// TwinCAT 3 PLC project VibrodriverPLC
// ProgramVersion: 3.1.4024.0
// libraries:
//   Tc2_MC2, * (Beckhoff Automation GmbH)
//   Tc2_NC, * (Beckhoff Automation GmbH)
//   Tc2_Standard, * (Beckhoff Automation GmbH)
//   Tc2_System, * (Beckhoff Automation GmbH)
//   Tc2_Utilities, * (Beckhoff Automation GmbH)
//   Tc3_Module, * (Beckhoff Automation GmbH)
//   VisuDialogs, * (System)
//   VisuSymbols,3.5.10.0,System
// project tree:
//   / GlobalTextList.TcGTLO, PlcTask.TcTTO, Visualization Manager.TcVMO (not stored)
//   POUs/ MAIN.TcPOU, FB_ReadGeophone.TcPOU, FB_ReadAccelerometer.TcPOU (not stored), P_ReadSensors.TcPOU (not stored)
//   VISUs/ hmi.TcVIS

CONFIGURATION VibrodriverPLC
    RESOURCE PLC ON TwinCAT3
        TASK PlcTask(INTERVAL := T#10ms, PRIORITY := 20);
        PROGRAM MAIN WITH PlcTask : MAIN;
        PROGRAM P_ReadSensors WITH PlcTask : P_ReadSensors;
    END_RESOURCE
END_CONFIGURATION

// ---- POUs/MAIN.TcPOU
PROGRAM MAIN
VAR

	bRun : BOOL := FALSE; // main control	

	axes : ARRAY[0..3] OF AXIS_REF; // [BL BR TL TR] (linked in MOTION)
	
	// motion control function blocks
	arrMCResets        		: ARRAY[0..3] OF MC_Reset;
	arrMCPowers				: ARRAY[0..3] OF MC_Power;
	arrMCSetPositions		: ARRAY[0..3] OF MC_SetPosition;
	arrMCMoveAbsolutes		: ARRAY[0..3] OF MC_MoveAbsolute;
	arrMCMoveRelatives		: ARRAY[0..3] OF MC_MoveRelative;
	arrMCMoveVelocitys 		: ARRAY[0..3] OF MC_MoveVelocity;
	arrMCHalts				: ARRAY[0..3] OF MC_Halt;
	arrMCGearIns			: ARRAY[1..3] OF MC_GearIn;
	arrMCGearOuts			: ARRAY[1..3] OF MC_GearOut;
	arrMCPhaseAbsolutes     : ARRAY[1..3] OF MC_PhasingAbsolute;
	
	arrRelsDone : ARRAY[0..3] OF BOOL; // keep track of if each motor is done its relative movement
	arrRelsDoneZero : ARRAY[0..3] OF BOOL; // keep track of if each motor is done its relative movement
	arrMCMoveRelativesZero	: ARRAY[0..3] OF MC_MoveRelative;
	arrZeroPoss : ARRAY[0..3] OF LREAL;
	
	arrHexErrors : ARRAY[0..3] OF T_MaxString; // store hex format of axes errors
	
	i: INT; // generic loop index 1
	j: INT; // generic loop index 2
	k: INT; // generic loop index 3
	
	bStarted : BOOL := FALSE; // if started is complete
	bCoupled : BOOL := FALSE;
	iMode : INT := 2; // 0 = move abs, 1 = move rel, 2 = move vel, 3 = zero nearest
	
	// button bools
	bStart  : BOOL := FALSE;
	bStop   : BOOL := TRUE;
	bCouple : BOOL := FALSE;
	bAbsPos : BOOL := FALSE;
	bRelPos	: BOOL := FALSE;
	bVel	: BOOL := TRUE;
	
	// taps
	bZeroNear : BOOL := FALSE;
	bResetFaults :BOOL := FALSE;
	
	// values in HMI
	iPos : INT := 0;
	iVel : INT := 1440;
	iAcc : INT := 720;
	iPhs : INT := 0;
	
	// track previous values for updating function blocks
	iPrevPos : INT := iPos;
	iPrevVel : INT := iVel;
	iPrevAcc : INT := iAcc;
	iPrevPhs : INT := iPhs;
	
	iMaxVel : INT := 3600; // max 10 hz
	eDirec : MC_Direction := MC_Direction.MC_Negative_Direction;
	iDirMult : INT := -1; // multiplier: actVel = setVel * mult (used to reverse default)
	
	// outside first and last are ignored
	iFirstIdx : INT := 2; // first motor index to control
	iLastIdx : INT := 3; // last motor index to control
	
	iEndIdx : INT := 3; // used to ignore other indices when the motors are coupled, set such that only the iFirstIdx index motor is controlled 
END_VAR

// test
FOR i := iFirstIdx TO iLastIdx DO
	// UPDATE AXES STATUS
	axes[i].ReadStatus();
	// UPDATE HEX ERRORS
	arrHexErrors[i] := WORD_TO_HEXSTR(in:=UDINT_TO_WORD(MAIN.axes[i].Status.ErrorID), iPrecision:=4, bLoCase:=FALSE);
	// RESTRICT VELOCITY
	IF ABS(axes[i].NcToPlc.ActVelo) > iMaxVel THEN
		M_SetState(0);
	END_IF
END_FOR


// STARTUP
// <<<<<<<<<<<<<<<<<<<<<<<<<<<<<<<<<<<<<<<<<<<<<<<<<<<<<<<
IF NOT bStarted THEN
	// start each motor
	FOR i := iFirstIdx TO iLastIdx DO
		// default to OFF despite variable values
		M_SetState(0);
		arrMCResets[i](Axis:=axes[i]);
		arrMCPowers[i](Axis:=axes[i], Enable:= TRUE, Enable_Positive:=TRUE, Enable_Negative:=TRUE);
	END_FOR
	
	// if all motors powered, set to started
	FOR i:=iFirstIdx TO iLastIdx DO
		IF NOT arrMCPowers[i].Status THEN
			EXIT;
		ELSIF i=iLastIdx THEN
			bStarted := TRUE;
			M_SetMode(2);
		END_IF
	END_FOR
END_IF
// >>>>>>>>>>>>>>>>>>>>>>>>>>>>>>>>>>>>>>>>>>>>>>>>>>>>>>>


// MODE SELECTION
// <<<<<<<<<<<<<<<<<<<<<<<<<<<<<<<<<<<<<<<<<<<<<<<<<<<<<<<
// prevent no mode selection
IF NOT bAbsPos AND iMode = 0 THEN
	bAbsPos := TRUE;
ELSIF NOT bRelPos AND iMode = 1 THEN
	bRelPos := TRUE;
ELSIF NOT bVel AND iMode = 2 THEN
	bVel := TRUE;
END_IF

// switch modes
IF iMode = 3 THEN
	M_SetMode(3);
ELSIF iMode = 4 THEN
	M_SetMode(4);
ELSIF bAbsPos AND iMode <> 0 THEN
	M_SetMode(0);
ELSIF bRelPos AND iMode <> 1 THEN
	M_SetMode(1);
ELSIF bVel AND iMode <> 2 THEN
	M_SetMode(2);
END_IF
// >>>>>>>>>>>>>>>>>>>>>>>>>>>>>>>>>>>>>>>>>>>>>>>>>>>>>>>


// RUN STATE SELECTION
// <<<<<<<<<<<<<<<<<<<<<<<<<<<<<<<<<<<<<<<<<<<<<<<<<<<<<<<
// prevent turning off a button, only swapping allowed
IF bRun AND NOT bStop THEN
	bStart := TRUE;
ELSIF NOT bRun AND NOT bStart THEN
	bStop := TRUE;
ELSE // invalid state
	bStop := TRUE;
END_IF

// on off logic
IF NOT bRun AND bStart THEN
	M_SetState(1);
END_IF
IF bStop THEN
	M_SetState(0);
END_IF

// handle zeroing button
IF bZeroNear AND NOT bRun THEN
	M_SetState(1);
	M_SetMode(3);
ELSIF bResetFaults AND NOT bRun THEN
	M_SetState(0);
	M_SetMode(4);
END_IF
// >>>>>>>>>>>>>>>>>>>>>>>>>>>>>>>>>>>>>>>>>>>>>>>>>>>>>>>


// COUPLING
// <<<<<<<<<<<<<<<<<<<<<<<<<<<<<<<<<<<<<<<<<<<<<<<<<<<<<<<
// disallow coupling while in motion
IF bCouple AND NOT bCoupled THEN
	FOR i:=iFirstIdx TO iLastIdx DO
		IF axes[i].Status.Moving THEN
			bCouple := FALSE;
			EXIT;
		END_IF
	END_FOR
END_IF

// COUPLE/UNCOUPLE GEARS
//arrMCGearOuts[1](Slave:=axes[1], Execute:=NOT bCouple AND bCoupled);
//arrMCGearOuts[2](Slave:=axes[2], Execute:=NOT bCouple AND bCoupled);
arrMCGearOuts[3](Slave:=axes[3], Execute:=NOT bCouple AND bCoupled);
//arrMCGearIns[1](Master:=axes[0], Slave:=axes[1], Execute:=bCouple AND NOT bCoupled, RatioNumerator:=-1);
//arrMCGearIns[2](Master:=axes[0], Slave:=axes[2], Execute:=bCouple AND NOT bCoupled, RatioNumerator:=-1);
arrMCGearIns[3](Master:=axes[2], Slave:=axes[3], Execute:=bCouple AND NOT bCoupled, RatioNumerator:=-1);

// check if uncoupling done
IF (NOT bCouple AND bCoupled)THEN
	FOR i:=iFirstIdx+1 TO iLastIdx DO
		IF NOT arrMCGearOuts[i].Done THEN
			EXIT;
		ELSIF i=iLastIdx THEN
			// if all out of gear, set the end index to the last index so that all the motors are controlled seperately again
			iEndIdx := iLastIdx;
			bCoupled := TRUE;
		END_IF;
	END_FOR
END_IF
// check if coupling done
IF (bCouple AND NOT bCoupled) THEN
	FOR i:=iFirstIdx+1 TO iLastIdx DO
		IF NOT arrMCGearIns[i].InGear THEN
			EXIT;
		ELSIF i=iLastIdx THEN
			// if all in gear, set the end index to the first index so that only the master is controlled
			iEndIdx := iFirstIdx;
			bCoupled := TRUE;
		END_IF;
	END_FOR
END_IF
// >>>>>>>>>>>>>>>>>>>>>>>>>>>>>>>>>>>>>>>>>>>>>>>>>>>>>>>





// operations to do only after startup
IF bStarted THEN
	

	// PHASING
	// set phase, master = BL, slave = TL
	// <<<<<<<<<<<<<<<<<<<<<<<<<<<<<<<<<<<<<<<<<<<<<<<<<<<<<<<
	
	IF iPrevPhs <> iPhs THEN
		//arrMCPhaseAbsolutes[1](Master:=axes[0], Slave:=axes[1], Execute:=FALSE); // set phase of BR w BL
		//arrMCPhaseAbsolutes[2](Master:=axes[0], Slave:=axes[2], Execute:=FALSE); // set phase of top w bottom
		arrMCPhaseAbsolutes[3](Master:=axes[2], Slave:=axes[3], Execute:=FALSE); // set phase of TR w TL
		iPrevPhs := iPhs;
	END_IF
	
	IF bRun AND bCoupled THEN
		// set phase of BR w BL
		//arrMCPhaseAbsolutes[1](Master:=axes[0], Slave:=axes[1], Execute:=TRUE, PhaseShift:=0, Velocity:=iVel+180);
		// set phase of top w bottom
		//arrMCPhaseAbsolutes[2](Master:=axes[0], Slave:=axes[2], Execute:=TRUE, PhaseShift:=iPhs, Velocity:=iVel+180);
		// set phase of TR w TL
		arrMCPhaseAbsolutes[3](Master:=axes[2], Slave:=axes[3], Execute:=TRUE, PhaseShift:=0, Velocity:=iVel+180);
	END_IF
	// >>>>>>>>>>>>>>>>>>>>>>>>>>>>>>>>>>>>>>>>>>>>>>>>>>>>>>>
	
	
	
	
	// MAIN COMMAND LOOP
	FOR i := iFirstIdx TO iEndIdx DO
		
	
		// CHANGE RESETING
		// <<<<<<<<<<<<<<<<<<<<<<<<<<<<<<<<<<<<<<<<<<<<<<<<<<<<<<<
		
		// if values have been updated, unexecute relevant functions so that they can restart with correct values
		IF (iPrevVel <> iVel) OR (iPrevAcc <> iAcc) THEN
			arrMCMoveAbsolutes[i](Axis:=axes[i], Execute:=FALSE);
			arrMCMoveRelatives[i](Axis:=axes[i], Execute:=FALSE);
			arrMCMoveVelocitys[i](Axis:=axes[i], Execute:=FALSE);
		ELSIF iPrevPos <> iPos THEN
			arrMCMoveAbsolutes[i](Axis:=axes[i], Execute:=FALSE);
			arrMCMoveRelatives[i](Axis:=axes[i], Execute:=FALSE);
		END_IF
		
		// if end index then set the previous values for change checks above ^
		IF i = iEndIdx THEN
			iPrevPos := iPos;
			iPrevVel := iVel;
			iPrevAcc := iAcc;
		END_IF
		// >>>>>>>>>>>>>>>>>>>>>>>>>>>>>>>>>>>>>>>>>>>>>>>>>>>>>>>
		
		
		// RELATIVE MOVEMENT OPERATION
		// <<<<<<<<<<<<<<<<<<<<<<<<<<<<<<<<<<<<<<<<<<<<<<<<<<<<<<<
		
		// check if relative movement is done, set to stop
		IF arrMCMoveRelatives[i].Done  THEN
			arrRelsDone[i] := TRUE;
			FOR j := iFirstIdx TO iEndIdx DO
				IF arrRelsDone[j] = FALSE THEN EXIT; END_IF
				IF j = iEndIdx THEN
					M_SetState(0);
					FOR k := iFirstIdx TO iLastIdx DO
						arrRelsDone[k] := FALSE;
					END_FOR
				END_IF
			END_FOR
		END_IF
		// check if relative movement is done, set to stop (SPECIFIC FOR ZEROING)
		IF arrMCMoveRelativesZero[i].Done  THEN
			arrRelsDoneZero[i] := TRUE;
			FOR j := iFirstIdx TO iEndIdx DO
				IF arrRelsDoneZero[j] = FALSE THEN EXIT; END_IF
				IF j = iEndIdx THEN
					M_SetState(0);
					FOR k := iFirstIdx TO iLastIdx DO
						arrRelsDoneZero[k] := FALSE;
					END_FOR
					IF iMode=3 THEN
						FOR k := iFirstIdx TO iLastIdx DO
							arrZeroPoss[k] := 0;
						END_FOR
						M_SetMode(2);
					END_IF
				END_IF
			END_FOR
		END_IF
		
		// calculate distance to nearest zero
		IF iMode = 3 AND arrZeroPoss[i] = 0 THEN
			IF axes[i].NcToPlc.ModuloActPos > 180 THEN
				arrZeroPoss[i] := 360 - axes[i].NcToPlc.ModuloActPos;
			ELSE
				arrZeroPoss[i] := -axes[i].NcToPlc.ModuloActPos;
			END_IF
		END_IF
		// >>>>>>>>>>>>>>>>>>>>>>>>>>>>>>>>>>>>>>>>>>>>>>>>>>>>>>>	
		
		
		
		
		// run MAIN OPERATIONS, execute values based on various bools
		// <<<<<<<<<<<<<<<<<<<<<<<<<<<<<<<<<<<<<<<<<<<<<<<<<<<<<<<
		
		arrMCSetPositions[i](Axis:=axes[i], Execute:=TRUE, Position:=0); // very important for some reason
		
		arrMCMoveAbsolutes[i](Axis:=axes[i], Execute:= iMode=0 AND bRun,
								Position:=iPos*iDirMult, Velocity:=iVel, Acceleration:=iAcc, Deceleration:=iAcc);
								
		arrMCMoveRelatives[i](Axis:=axes[i], Execute:= iMode=1 AND bRun AND NOT arrRelsDone[i],
								Distance:=iPos*iDirMult, Velocity:=iVel, Acceleration:=iAcc, Deceleration:=iAcc);
								
		arrMCMoveVelocitys[i](Axis:=axes[i], Execute:= iMode=2 AND bRun, Direction:=eDirec,
								Velocity:=iVel, Acceleration:=iAcc, Deceleration:=iAcc);
								
		arrMCMoveRelativesZero[i](Axis:=axes[i], Execute:= iMode=3 AND bRun AND NOT arrRelsDoneZero[i],
								Distance:=arrZeroPoss[i], Velocity:=iVel, Acceleration:=iAcc, Deceleration:=iAcc);
		
		// NEVER MOVE FROM LAST CALL
		arrMCHalts[i](Axis:=axes[i],Execute:=NOT bRun, Deceleration:=400);
		// >>>>>>>>>>>>>>>>>>>>>>>>>>>>>>>>>>>>>>>>>>>>>>>>>>>>>>>	
	END_FOR
END_IF

METHOD PRIVATE M_SetMode
VAR_INPUT
	iModeSet : INT;
END_VAR
CASE iModeSet OF
	0 : // move absolute
		bAbsPos := TRUE;
		bRelPos := FALSE;
		bVel := FALSE;
		iMode := 0;
	1 : // move relative
		bAbsPos := FALSE;
		bRelPos := TRUE;
		bVel := FALSE;
		iMode := 1;
	2 : // move velocity
		bAbsPos := FALSE;
		bRelPos := FALSE;
		bVel := TRUE;
		iMode := 2;
	3 : // move to nearest zero
		bAbsPos := FALSE;
		bRelPos := FALSE;
		bVel := FALSE;
		iMode := 3;
	
	4 : // reset faults
		bAbsPos := FALSE;
		bRelPos := FALSE;
		bVel := FALSE;
		iMode := 4;
		bStarted := FALSE;
	ELSE
		ADSLOGSTR(
			msgCtrlMask := ADSLOG_MSGTYPE_ERROR, 
			msgFmtStr   := 'Invalid Mode%s', 
			strArg      := ''
		); 
END_CASE
END_METHOD

METHOD PRIVATE M_SetState
VAR_INPUT
	iState: INT;
END_VAR
CASE iState OF
	0 :
		bRun := FALSE;
		bStart := FALSE;
		bStop := TRUE;
	1 :
		bRun := TRUE;
		bStart := TRUE;
		bStop := FALSE;
	ELSE
		ADSLOGSTR(
			msgCtrlMask := ADSLOG_MSGTYPE_ERROR, 
			msgFmtStr   := 'Invalid State%s', 
			strArg      := ''
		); 
END_CASE
END_METHOD

END_PROGRAM

// ---- POUs/FB_ReadGeophone.TcPOU
FUNCTION_BLOCK FB_ReadGeophone
VAR_INPUT
	// none
END_VAR
VAR_OUTPUT
	velX : LREAL; // left -> right
	velY : LREAL; // back -> front
	velZ : LREAL; // top -> bottom
END_VAR
VAR
	c1Sample AT %I* : DINT; // channel 1 voltage (mV) -  x axis (yellow arrow)
	c2Sample AT %I* : DINT; // channel 2 voltage (mV) -  y axis (red arrow)
	c3Sample AT %I* : DINT; // channel 3 voltage (mV) -  z axis (rods -> level)
	
	// all real since need to be converted anyway
	peakVal : REAL := 10;
	maxInt : REAL := 7812500;
	sens : REAL := 78.9; // volts per meter per second
	unitMult : REAL := 1000; // m/s to mm/s
	mult : REAL := peakVal / maxInt / sens * unitMult;
END_VAR


// m/s
velX := DINT_TO_REAL(c1Sample) * mult;
velY := DINT_TO_REAL(c2Sample) * mult;
velZ := DINT_TO_REAL(c3Sample) * mult;

END_FUNCTION_BLOCK

// ---- GlobalTextList.TcGTLO
TEXTLIST GlobalTextList
  610 = '%.0f'
  395 = '%.Of'
  543 = '%s'
  196 = '0'
  727 = 'Abs. Position'
  848 = 'Abs. Position:'
  942 = 'Acceleration'
  31 = 'Acceleration:'
  909 = 'BL'
  278 = 'BL Torque:'
  207 = 'BR'
  495 = 'BR Torque:'
  18 = 'Couple'
  782 = 'COUPLE'
  471 = 'Error #'
  37 = 'Labelhttps://infosys.beckhoff.com/english.php?https://infosys.beckhoff.com/english.php?content=../content/1033/tcncerrcode2/513133323.html&id='
  295 = 'Mode'
  778 = 'Movement Mode'
  187 = 'Phase'
  200 = 'Phase:'
  572 = 'Position'
  777 = 'Position Target'
  556 = 'Position:'
  61 = 'Rel. Position:'
  4 = 'Rel. Positon'
  553 = 'Rel. Velocity:'
  359 = 'Reset Faults'
  245 = 'Run Mode'
  864 = 'Set Phase'
  421 = 'Setpoints'
  792 = 'START'
  174 = 'STOP'
  592 = 'TL'
  858 = 'TL Torque:'
  531 = 'TR'
  672 = 'TR Torque:'
  226 = 'U/L Phase:'
  770 = 'Velocity'
  275 = 'Velocity:'
  935 = 'Vibrodriver HMI'
  169 = 'x%s'
  868 = 'xs'
  875 = 'Zero to Nearest'
END_TEXTLIST

// ---- VISUs/hmi.TcVIS
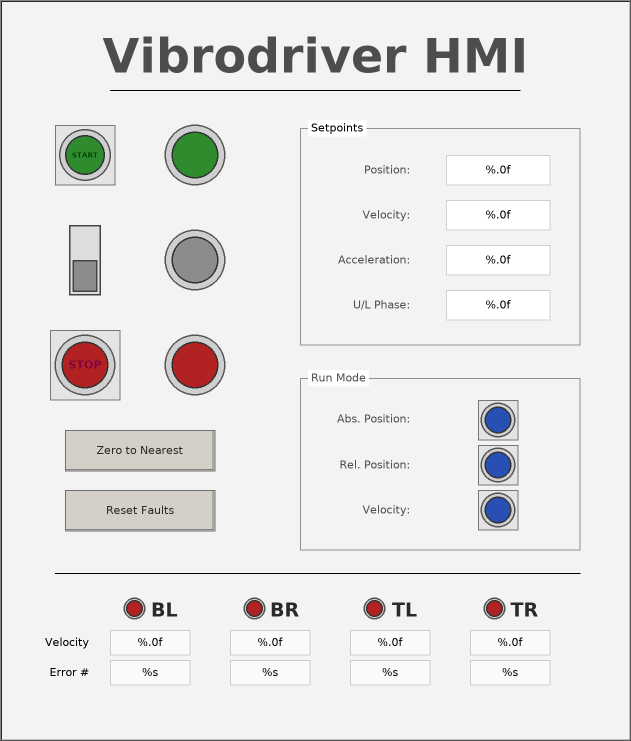
VISUALIZATION hmi  // 631x741
    RoundedRectangle (0,0 631x741)
    PushSwitch (55,125 60x60), tooltip "START", variable: MAIN.bStart, behaviour: TOGGLE, style: Switch-PushSwitch-Green
    Lamp1 (160,120 70x70), variable: MAIN.bStart, style: Lamp-Lamp1-Green
    PushSwitch (50,330 70x70), tooltip "STOP", variable: MAIN.bStop, behaviour: TOGGLE, style: Switch-PushSwitch-Red
    Lamp1 (160,330 70x70), variable: MAIN.bStop, style: Lamp-Lamp1-Red
    GroupBox (300,120 280x225), "Setpoints"
        Label (16,80 97x30), "Velocity:"
        Label (16,125 97x30), "Acceleration:"
        Textfield (146,80 104x30), "%.0f", text variable: MAIN.iVel
            OnMouseClick: write the text variable via InputWithLimits, min -(MAIN.iMaxVel - 200), max MAIN.iMaxVel - 200, format %d
        Textfield (146,35 104x30), "%.0f", text variable: MAIN.iPos
            OnMouseClick: write the text variable via InputWithLimits
        Textfield (146,125 104x30), "%.0f", text variable: MAIN.iAcc
            OnMouseClick: write the text variable via InputWithLimits, min 0, format %d
        Label (16,35 97x30), "Position:"
        Label (16,170 97x30), "U/L Phase:"
        Textfield (146,170 104x30), "%.0f", text variable: MAIN.iPhs
            OnMouseClick: write the text variable via InputWithLimits, min -360, max 360, format %d
    GroupBox (300,370 280x180), "Run Mode"
        Label (16,80 97x30), "Rel. Position:"
        Label (16,125 97x30), "Velocity:"
        Label (16,34 97x30), "Abs. Position:"
        PushSwitch (178,30 40x40), variable: MAIN.bAbsPos, behaviour: TOGGLE, style: Switch-PushSwitch-Blue
        PushSwitch (178,75 40x40), variable: MAIN.bRelPos, behaviour: TOGGLE, style: Switch-PushSwitch-Blue
        PushSwitch (178,120 40x40), variable: MAIN.bVel, behaviour: TOGGLE, style: Switch-PushSwitch-Blue
    DipSwitch (50,225 70x70), tooltip "COUPLE", variable: MAIN.bCouple, behaviour: TOGGLE, style: Switch-DipSwitch-Gray
    Lamp1 (160,225 70x70), variable: MAIN.bCouple, style: Lamp-Lamp1-Gray
    Label (60,350 50x30), "STOP"
    Label (60,140 50x30), "START"
    Button (65,430 150x41), "Zero to Nearest"
        tap MAIN.bZeroNear
    Label (50,20 531x71), "Vibrodriver HMI"
    Line (110,90) (520,90)
    Label (242,590 85x40), "BR"
    Label (362,590 85x40), "TL"
    Label (482,590 85x40), "TR"
    Button (65,490 150x41), "Reset Faults"
        tap MAIN.bResetFaults
    Label (122,590 85x40), "BL"
    Line (55,573) (580,573)
    Lamp1 (122,596 25x25), variable: MAIN.axes[0].Status.Error, style: Lamp-Lamp1-Red
    Lamp1 (242,596 25x25), variable: MAIN.axes[1].Status.Error, style: Lamp-Lamp1-Red
    Lamp1 (482,596 25x25), variable: MAIN.axes[3].Status.Error, style: Lamp-Lamp1-Red
    Lamp1 (362,596 25x25), variable: MAIN.axes[2].Status.Error, style: Lamp-Lamp1-Red
    Textfield (110,630 80x25), "%.0f", text variable: MAIN.axes[0].NcToPlc.ActVelo
    Textfield (230,630 80x25), "%.0f", text variable: MAIN.axes[1].NcToPlc.ActVelo
    Textfield (350,630 80x25), "%.0f", text variable: MAIN.axes[2].NcToPlc.ActVelo
    Textfield (470,630 80x25), "%.0f", text variable: MAIN.axes[3].NcToPlc.ActVelo
    Textfield (110,660 80x25), "%s", text variable: MAIN.arrHexErrors[0]
    Textfield (230,660 80x25), "%s", text variable: MAIN.arrHexErrors[1]
    Textfield (350,660 80x25), "%s", text variable: MAIN.arrHexErrors[2]
    Textfield (470,660 80x25), "%s", text variable: MAIN.arrHexErrors[3]
    Label (40,660 52x25), "Error #"
    Label (40,630 52x25), "Velocity"
END_VISUALIZATION
